TYPE strRecivedata :
	STRUCT
		arbyDATA	: ARRAY[0..Sewts_TCP.MAX_Bool_SIZE] OF BOOL;   											(*Job done *)	
	END_STRUCT
END_TYPE

(* stored: Version 1.1.0.1, ProductVersion 3.1.4024.12
   DUT strRecivedata: Id {77127be8-197e-460e-8a10-0b2b0a7588f9} *)
